(* CoDeSys 2.3.9.44 project: Cap11_17.pro *)
(* Libraries: Standard.lib 4.10.05 10:14:46, IecSfc.lib 13.4.06 14:51:28 *)

(* Task configuration *)
TASK NewTask (PRIORITY := 1, INTERVAL := T#100ms);
	PLC_PRG
END_TASK

(* Global variable list: Global_Variables *)
VAR_GLOBAL
    (* Entradas*)
    LInf: BOOL;
    LSup:BOOL;
    PS1:BOOL;
    PS2:BOOL;
    M:BOOL;

   (* Salidas *)
   V1:BOOL;
   V2:BOOL;
   VA:BOOL;
   VB:BOOL;
   VC:BOOL;
   Motor:BOOL;
END_VAR

(* POU PLC_PRG, ST *)
PROGRAM PLC_PRG
VAR
END_VAR
Depositos;
Automatismo;
END_PROGRAM

(* POU Depositos, ST *)
PROGRAM Depositos
VAR
   Nivel: REAL:=0.2;
   ValvulaEntrada:BOOL;
   ValvulaSalida:BOOL;
   CaudalEntrada:REAL:=0;
   CaudalSalida:REAL:=0;
   Area:REAL:=1;
   IntT:REAL:=0.1;
   KEntrada:REAL:=0.3;
   KSalida:REAL:=0.4;
	Neto: REAL;
	Nivellnf:REAL:=0;
	NivelSup:REAL:=2.2;
	CaudalEntrada2: REAL;
	CaudalSalida2: REAL;
	Neto2: REAL;
	Nivel2: REAL;
	Nivellnf2: REAL:=0;
	NivelSup2: REAL:=4;
	KSalida2: REAL:=0.8;
END_VAR
(*Deposito 1 *)
CaudalEntrada:=BOOL_TO_INT(V1)*KEntrada;
CaudalSalida:=BOOL_TO_INT(V2)*KSalida;
Neto:=(CaudalEntrada-CaudalSalida);
IF (Neto<0AND Nivel>Nivellnf) OR (Neto>0 AND Nivel<NivelSup) THEN
   Nivel:=Nivel+IntT*Neto;
END_IF

IF Nivel>0.33 THEN
   LInf:=TRUE;
ELSE
   LInf:=FALSE;
END_IF

IF Nivel>1.85 THEN
   LSup:=TRUE;
ELSE
   LSup:=FALSE;
END_IF

(*Deposito 2 *)
CaudalEntrada2:=(BOOL_TO_INT(VA)+BOOL_TO_INT(VB))*KEntrada;
CaudalSalida2:=BOOL_TO_INT(VC)*KSalida2;
Neto2:=(CaudalEntrada2-CaudalSalida2);
IF (Neto2<0AND Nivel2>Nivellnf2) OR (Neto2>0 AND Nivel2<NivelSup2) THEN
   Nivel2:=Nivel2+IntT*Neto2;
END_IF


IF Nivel2>2 THEN
   PS1:=TRUE;
ELSE
   PS1:=FALSE;
END_IF

IF Nivel2>3 THEN
   PS2:=TRUE;
ELSE
   PS2:=FALSE;
END_IF
END_PROGRAM

(* POU Automatismo, SFC *)
PROGRAM Automatismo
VAR
END_VAR
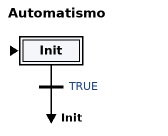
INITIAL_STEP Init:
END_STEP
TRANSITION FROM Init TO Init := TRUE;
END_TRANSITION
END_PROGRAM

(* Visualisation Deposito
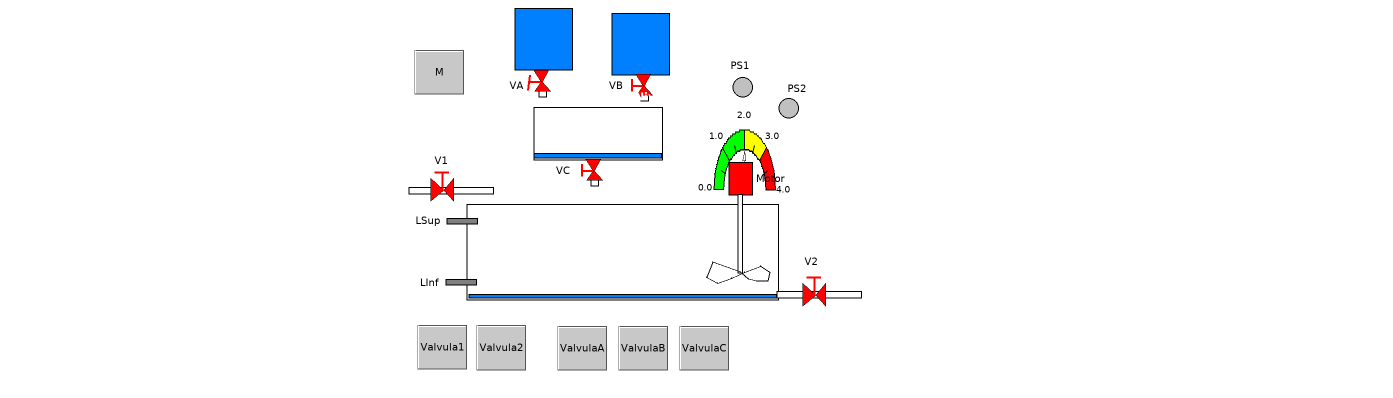
button at (30,345)-(79,389): text "Valvula1"; toggles V1
button at (89,345)-(138,390): text "Valvula2"; toggles V2
rectangle at (81,314)-(389,318): top -40*Depositos.Nivel
rectangle at (389,311)-(474,318): alarm colour if Valvula2 AND Depositos.Nivel>0
rectangle at (21,207)-(106,214): alarm colour if Valvula1
polygon at (415,303)-(428,326): alarm colour if V2
polygon at (428,303)-(438,326): alarm colour if V2
polyline at (427,297)-(427,314): alarm colour if V2
polyline at (419,297)-(433,297): alarm colour if V2
rectangle at (59,238)-(90,244): alarm colour if LSup
rectangle at (58,299)-(89,305): alarm colour if LInf
polygon at (248,94)-(263,105): alarm colour if VB
polygon at (249,105)-(265,115): alarm colour if VB
polyline at (244,106)-(255,106): alarm colour if VB
polyline at (244,99)-(244,111): alarm colour if VB
button at (170,346)-(219,390): text "ValvulaA"; toggles VA
button at (231,346)-(280,390): text "ValvulaB"; toggles VB
polygon at (198,179)-(213,190): alarm colour if VC
polygon at (199,190)-(215,200): alarm colour if VC
polyline at (194,191)-(205,191): alarm colour if VC
polyline at (194,184)-(194,196): alarm colour if VC
button at (292,346)-(341,390): text "ValvulaC"; toggles VC
rectangle at (146,173)-(274,178): top -10*Depositos.Nivel2
group at (308,116)-(405,223)
  rectangle at (0,0)-(1,1): text "{ExtendedElement},Visu\ElementDLL.ete,0,@Zeigerinstrument,97,180,0,0,255,255,255,0,Depositos.Nivel2,,%.1f,0,1,1,0.5,1,0,4,0,0,0,0,0,0,0,-11,80,400,Arial,1,3,0,2,0,255,0,2,3,255,255,0,3,4,255,0,0,0,255,255,255,,0,0,0,0,"
  rectangle at (0,41)-(19,55): text "0.0"
  rectangle at (11,14)-(30,28): text "1.0"
  rectangle at (39,3)-(58,17): text "2.0"
  rectangle at (67,14)-(86,28): text "3.0"
  rectangle at (78,42)-(97,56): text "4.0"
  polygon at (47,29)-(50,49): angle ((Depositos.Nivel2 * 1.0)-2) * 45
ellipse at (345,97)-(365,117): alarm colour if PS1
ellipse at (391,118)-(411,138): alarm colour if PS2
rectangle at (35,165)-(72,196): text "V1"
rectangle at (405,266)-(442,297): text "V2"
rectangle at (110,90)-(147,121): text "VA"
rectangle at (210,90)-(247,121): text "VB"
rectangle at (157,175)-(194,206): text "VC"
rectangle at (334,70)-(371,101): text "PS1"
rectangle at (391,93)-(428,124): text "PS2"
rectangle at (23,287)-(60,318): text "LInf"
rectangle at (22,225)-(59,256): text "LSup"
rectangle at (341,182)-(365,215): alarm colour if Motor
rectangle at (364,183)-(401,214): text "Motor"
button at (27,70)-(76,114): text "M"; taps M
polygon at (43,198)-(56,221): alarm colour if V1
polygon at (56,198)-(66,221): alarm colour if V1
polyline at (55,192)-(55,209): alarm colour if V1
polyline at (47,192)-(61,192): alarm colour if V1
polygon at (146,90)-(161,101): alarm colour if VA
polygon at (147,101)-(163,111): alarm colour if VA
polyline at (142,102)-(153,102): alarm colour if VA
polyline at (140,95)-(142,110): alarm colour if VA
25 more shapes without text or variables
*)
